{attribute 'Tc2GvlVarNames'}
VAR_CONFIG
END_VAR

(* stored: Version 1.1.0.1, ProductVersion 3.1.0.26
   GVL Variable_Configuration: Id {e06bac96-a6ca-40e8-a2dd-6d60c8bf7be0} *)
